// TIA Portal V16 export
// export: Created 2022-11-17T15:49:32.5672414Z, ExportSetting WithDefaults, DisplayName Totally Integrated Automation Portal, DisplayVersion V16 Update 6, DisplayName TIA Portal Version Control Interface, DisplayVersion V16 Update 2, DisplayName TIA Portal Openness, DisplayVersion V16 Update 6, DisplayName SINAMICS Startdrive Advanced, DisplayVersion V16 Update 5, DisplayName SINAMICS Startdrive G130, G150, S120, S150, SINAMICS MV, S210, DisplayVersion V16 Update 5, DisplayName SINAMICS Startdrive G110M, G120, G120C, G120D, G120P, G115D, DisplayVersion V16 Update 5, DisplayName STEP 7 Professional, DisplayVersion V16 Update 6, DisplayName STEP 7 Safety, DisplayVersion V16, DisplayName WinCC Advanced, DisplayVersion V16 Update 6
FUNCTION "FC310_Motors" : Void   // FC310, LAD
{ S7_Optimized_Access := 'TRUE' }
VERSION : 0.1
// stored: AutoNumber false, IsIECCheckEnabled false, SetENOAutomatically false, UDAEnableTagReadback false
   VAR_INPUT
      Motor : Int;   // 0=NO; 1=Arm; 2=Carr; 3=Prestretch; 4=Stretch; 5=SX; 6=CM; 7=DX; 8=Top
      Dir : Bool;   // 0=BKWD; 1=FWD
      Start : Bool;
      Setpoint : Int;
   END_VAR
   VAR_TEMP
      SP_real : Real;
      Carr_Dec_low : DInt;
      Carr_Dec_high : DInt;
   END_VAR
   VAR_TEMP   // added for the SCL form of the ladder/FBD networks
      _w1 : Bool;
      _w2 : Bool;
      _w3 : Bool;
   END_VAR
BEGIN

REGION Network 1: Setpoint conversion
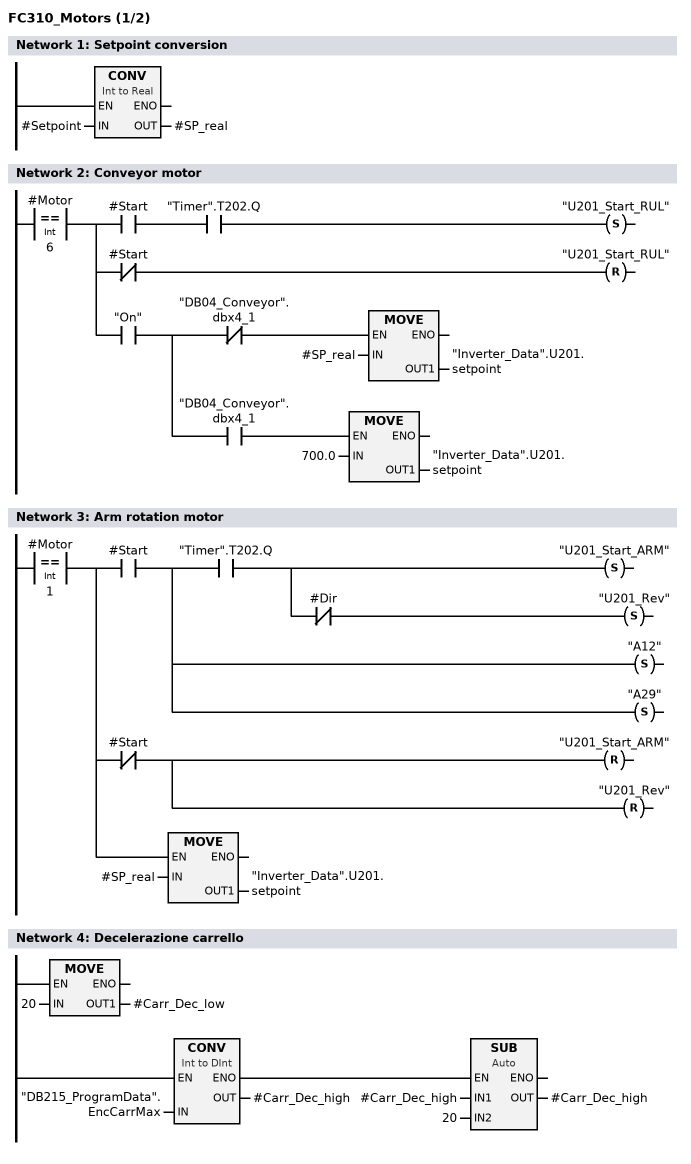
   RUNG wire#powerrail
      { S7_Templates := "[SrcType := Int, DestType := Real]" } Convert(in := #Setpoint, out => #SP_real)
   END_RUNG
   // the same network as SCL:
   #SP_real := INT_TO_REAL(#Setpoint);
END_REGION

REGION Network 2: Conveyor motor
   RUNG wire#powerrail
      { S7_Templates := "SrcType := Int" } EQ_Contact(in1 := #Motor, in2 := 6)
      wire#w1
      Contact( #Start )
      Contact( "Timer".T202.Q )
      S_Coil( "U201_Start_RUL" )
   END_RUNG
   RUNG wire#w1
      I_Contact( #Start )
      R_Coil( "U201_Start_RUL" )
   END_RUNG
   RUNG wire#w1
      Contact( "On" )
      wire#w2
      I_Contact( "DB04_Conveyor".dbx4_1 )
      Move(in := #SP_real, out1 => "Inverter_Data".U201.setpoint)
   END_RUNG
   RUNG wire#w2
      Contact( "DB04_Conveyor".dbx4_1 )
      Move(in := 700.0, out1 => "Inverter_Data".U201.setpoint)
   END_RUNG
   // the same network as SCL:
   #_w1 := #Motor = 6;
   IF #_w1 AND #Start AND "Timer".T202.Q THEN "U201_Start_RUL" := TRUE; END_IF;
   IF #_w1 AND NOT #Start THEN "U201_Start_RUL" := FALSE; END_IF;
   #_w2 := #_w1 AND "On";
   IF #_w2 AND NOT "DB04_Conveyor".dbx4_1 THEN "Inverter_Data".U201.setpoint := #SP_real; END_IF;
   IF #_w2 AND "DB04_Conveyor".dbx4_1 THEN "Inverter_Data".U201.setpoint := 700.0; END_IF;
END_REGION

REGION Network 3: Arm rotation motor
   RUNG wire#powerrail
      { S7_Templates := "SrcType := Int" } EQ_Contact(in1 := #Motor, in2 := 1)
      wire#w1
      Contact( #Start )
      wire#w2
      Contact( "Timer".T202.Q )
      wire#w3
      S_Coil( "U201_Start_ARM" )
   END_RUNG
   RUNG wire#w3
      I_Contact( #Dir )
      S_Coil( "U201_Rev" )
   END_RUNG
   RUNG wire#w2
      S_Coil( "A12" )
   END_RUNG
   RUNG wire#w2
      S_Coil( "A29" )
   END_RUNG
   RUNG wire#w1
      I_Contact( #Start )
      wire#w4
      R_Coil( "U201_Start_ARM" )
   END_RUNG
   RUNG wire#w4
      R_Coil( "U201_Rev" )
   END_RUNG
   RUNG wire#w1
      Move(in := #SP_real, out1 => "Inverter_Data".U201.setpoint)
   END_RUNG
   // the same network as SCL:
   #_w1 := #Motor = 1;
   #_w2 := #_w1 AND #Start;
   #_w3 := #_w2 AND "Timer".T202.Q;
   IF #_w3 THEN "U201_Start_ARM" := TRUE; END_IF;
   IF #_w3 AND NOT #Dir THEN "U201_Rev" := TRUE; END_IF;
   IF #_w2 THEN
       "A12" := TRUE;
       "A29" := TRUE;
   END_IF;
   IF #_w1 AND NOT #Start THEN
       "U201_Start_ARM" := FALSE;
       "U201_Rev" := FALSE;
   END_IF;
   IF #_w1 THEN "Inverter_Data".U201.setpoint := #SP_real; END_IF;
END_REGION

REGION Network 4: Decelerazione carrello
   RUNG wire#powerrail
      Move(in := 20, out1 => #Carr_Dec_low)
   END_RUNG
   RUNG wire#powerrail
      { S7_Templates := "[SrcType := Int, DestType := DInt]" } Convert(in := "DB215_ProgramData".EncCarrMax, out => #Carr_Dec_high)
      Sub(in1 := #Carr_Dec_high, in2 := 20, out => #Carr_Dec_high)
   END_RUNG
   // the same network as SCL:
   #Carr_Dec_low := 20;
   #Carr_Dec_high := INT_TO_DINT("DB215_ProgramData".EncCarrMax);
   #Carr_Dec_high := #Carr_Dec_high - 20;
END_REGION

REGION Network 5: Carriage motor
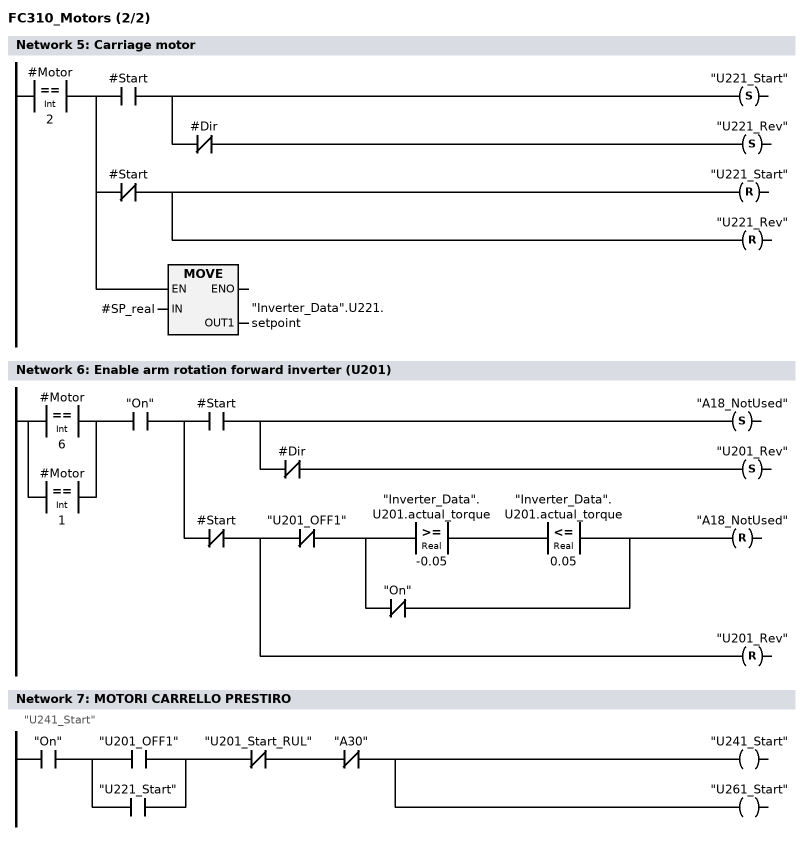
   RUNG wire#powerrail
      { S7_Templates := "SrcType := Int" } EQ_Contact(in1 := #Motor, in2 := 2)
      wire#w1
      Contact( #Start )
      wire#w2
      S_Coil( "U221_Start" )
   END_RUNG
   RUNG wire#w2
      I_Contact( #Dir )
      S_Coil( "U221_Rev" )
   END_RUNG
   RUNG wire#w1
      I_Contact( #Start )
      wire#w3
      R_Coil( "U221_Start" )
   END_RUNG
   RUNG wire#w3
      R_Coil( "U221_Rev" )
   END_RUNG
   RUNG wire#w1
      Move(in := #SP_real, out1 => "Inverter_Data".U221.setpoint)
   END_RUNG
   // the same network as SCL:
   #_w1 := #Motor = 2;
   #_w2 := #_w1 AND #Start;
   IF #_w2 THEN "U221_Start" := TRUE; END_IF;
   IF #_w2 AND NOT #Dir THEN "U221_Rev" := TRUE; END_IF;
   IF #_w1 AND NOT #Start THEN
       "U221_Start" := FALSE;
       "U221_Rev" := FALSE;
   END_IF;
   IF #_w1 THEN "Inverter_Data".U221.setpoint := #SP_real; END_IF;
END_REGION

REGION Network 6: Enable arm rotation forward inverter (U201)
   RUNG wire#powerrail
      { S7_Templates := "SrcType := Int" } EQ_Contact(in1 := #Motor, in2 := 6)
      wire#w1
      Contact( "On" )
      wire#w2
      Contact( #Start )
      wire#w3
      S_Coil( "A18_NotUsed" )
   END_RUNG
   RUNG wire#powerrail
      { S7_Templates := "SrcType := Int" } EQ_Contact(in1 := #Motor, in2 := 1)
   END_RUNG wire#w1
   RUNG wire#w3
      I_Contact( #Dir )
      S_Coil( "U201_Rev" )
   END_RUNG
   RUNG wire#w2
      I_Contact( #Start )
      wire#w4
      I_Contact( "U201_OFF1" )
      wire#w5
      { S7_Templates := "SrcType := Real" } GE_Contact(in1 := "Inverter_Data".U201.actual_torque, in2 := -0.05)
      { S7_Templates := "SrcType := Real" } LE_Contact(in1 := "Inverter_Data".U201.actual_torque, in2 := 0.05)
      wire#w6
      R_Coil( "A18_NotUsed" )
   END_RUNG
   RUNG wire#w5
      I_Contact( "On" )
   END_RUNG wire#w6
   RUNG wire#w4
      R_Coil( "U201_Rev" )
   END_RUNG
   // the same network as SCL:
   #_w1 := ((#Motor = 6) OR (#Motor = 1)) AND "On";
   #_w2 := #_w1 AND #Start;
   IF #_w2 THEN "A18_NotUsed" := TRUE; END_IF;
   IF #_w2 AND NOT #Dir THEN "U201_Rev" := TRUE; END_IF;
   #_w3 := #_w1 AND NOT #Start;
   IF #_w3 AND NOT "U201_OFF1" AND ((("Inverter_Data".U201.actual_torque >= (-0.05)) AND ("Inverter_Data".U201.actual_torque <= 0.05)) OR NOT "On") THEN
       "A18_NotUsed" := FALSE;
   END_IF;
   IF #_w3 THEN "U201_Rev" := FALSE; END_IF;
END_REGION

REGION Network 7: MOTORI CARRELLO PRESTIRO
   // "U241_Start"
   RUNG wire#powerrail
      Contact( "On" )
      wire#w1
      Contact( "U201_OFF1" )
      wire#w2
      I_Contact( "U201_Start_RUL" )
      I_Contact( "A30" )
      wire#w3
      Coil( "U241_Start" )
   END_RUNG
   RUNG wire#w1
      Contact( "U221_Start" )
   END_RUNG wire#w2
   RUNG wire#w3
      Coil( "U261_Start" )
   END_RUNG
   // the same network as SCL:
   "U241_Start" := "On" AND ("U201_OFF1" OR "U221_Start") AND NOT "U201_Start_RUL" AND NOT "A30";
   "U261_Start" := "U241_Start";
END_REGION
END_FUNCTION
